FUNCTION FIELDBUS_WORD_TO_PERCENT
  (* Standard: 61499-1 *)
  (* Version 1.0, 2023-10-21, franz *)
  PACKAGE signalprocessing;
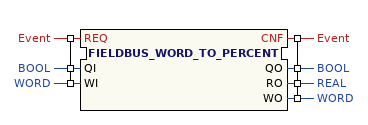
  EVENT_INPUT
    REQ WITH QI, WI;
  END_EVENT
  EVENT_OUTPUT
    CNF WITH QO, RO, WO;
  END_EVENT
  VAR_INPUT
    QI : BOOL;
    WI : WORD;
  END_VAR
  VAR_OUTPUT
    QO : BOOL;
    RO : REAL;
    WO : WORD;
  END_VAR
  BODY IN ST:
PACKAGE signalprocessing;

FUNCTION FIELDBUS_WORD_TO_PERCENT
VAR_INPUT
	QI : BOOL;
	WI : WORD;
END_VAR

VAR_OUTPUT
	QO : BOOL;
	RO : REAL;
	WO : WORD;
END_VAR

QO := QI;
IF (TRUE = QI) THEN
	IF (WI <= FIELDBUS_VALID_SIGNAL_W) THEN
		WO := WI;
		RO := UDINT_TO_REAL(WORD_TO_UDINT(WO)) / UDINT_TO_REAL(WORD_TO_UDINT(FIELDBUS_VALID_SIGNAL_W));
	END_IF;
END_IF;
END_FUNCTION
  END_BODY
END_FUNCTION
